(* PLC project turret, Dassault Systèmes ControlBuild 2024x Refresh1 *)
(* stored: creationDateTime 2024-01-23T17:34:07-01:00 *)

CONFIGURATION turret
  VAR_GLOBAL
    simuperiod : REAL := 50000.0;
    taskname : STRING(50) := 'turret.exe';
    allowpreconditions : BOOL := true;
    allowpostconditions : BOOL := true;
  END_VAR
END_CONFIGURATION
